Fanuc KAREL source: RSET_INT_REG.kl

PROGRAM T
%NOLOCKGROUP
VAR
 v0 : STRING[40]
 v1 : BOOLEAN
 v2 : INTEGER
 v3 : INTEGER
BEGIN
 RSET_INT_REG(v0, v1, v2, v3)
END T
